ArrayBool_TO_ArrayByte(ADR(GVL_IO.Q_Temp),SIZEOF(GVL_IO.Q_Temp),ADR(GVL_IO.Q),SIZEOF(GVL_IO.Q));
ArrayByte_TO_ArrayBool(ADR(GVL_IO.I),SIZEOF(GVL_IO.I),ADR(GVL_IO.I_Temp),SIZEOF(GVL_IO.I_Temp));




// IO屏蔽
IF GVL_Data.stRecipe.eMachineType<>_eMachineType THEN
	_boolTemp:=ADR(GVL.stShield_I);
	FOR _i:=0 TO SIZEOF(GVL.stShield_I)-1 BY 1 DO
		_boolTemp[_i]:=FALSE;
	END_FOR
	_boolTemp:=ADR(GVL.stShield_Q);
	FOR _i:=0 TO SIZEOF(GVL.stShield_Q)-1 BY 1 DO
		_boolTemp[_i]:=FALSE;
	END_FOR
	_eMachineType:=GVL_Data.stRecipe.eMachineType;
END_IF



CASE GVL_Data.stRecipe.eMachineType OF
	E_MachineType._200:
		GVL.stShield_I[0,5]:=TRUE;		
		GVL.stShield_I[0,6]:=TRUE;		
		GVL.stShield_I[0,7]:=TRUE;		
		GVL.stShield_I[0,8]:=TRUE;		
		GVL.stShield_I[0,9]:=TRUE;		
		GVL.stShield_I[0,10]:=TRUE;		
		GVL.stShield_I[0,11]:=TRUE;		
		GVL.stShield_I[0,12]:=TRUE;	
		GVL.stShield_I[3,10]:=TRUE;
		GVL.stShield_I[3,11]:=TRUE;
		GVL.stShield_I[3,12]:=TRUE;
		GVL.stShield_I[3,13]:=TRUE;
		GVL.stShield_I[6,14]:=TRUE;
		
		GVL.stShield_Q[0,7]:=TRUE;
		GVL.stShield_Q[0,12]:=TRUE;
		GVL.stShield_Q[0,13]:=TRUE;
		GVL.stShield_Q[3,10]:=TRUE;
		GVL.stShield_Q[3,11]:=TRUE;
		GVL.stShield_Q[3,12]:=TRUE;
		GVL.stShield_Q[3,13]:=TRUE;
		GVL.stShield_Q[5,11]:=TRUE;
		
		FOR _i:=0 TO 15 BY 1 DO
			GVL.stShield_I[7,_i]:=TRUE;
			GVL.stShield_Q[6,_i]:=TRUE;
		END_FOR
	E_MachineType._367:
		FOR _i:=6 TO 15 BY 1 DO
			GVL.stShield_I[1,_i]:=TRUE;
			GVL.stShield_Q[1,_i]:=TRUE;
		END_FOR
	
		GVL.stShield_I[0,5]:=TRUE;		
		GVL.stShield_I[0,6]:=FALSE;		
		GVL.stShield_I[0,7]:=TRUE;				
		GVL.stShield_I[0,10]:=TRUE;		
		GVL.stShield_I[0,11]:=TRUE;		
		GVL.stShield_I[0,12]:=FALSE;	
		GVL.stShield_I[0,13]:=TRUE;
		GVL.stShield_I[0,14]:=TRUE;
		GVL.stShield_I[0,15]:=TRUE;
		GVL.stShield_I[3,14]:=TRUE;
		GVL.stShield_I[3,15]:=TRUE;
		GVL.stShield_I[4,0]:=TRUE;
		GVL.stShield_I[4,1]:=TRUE;
		GVL.stShield_I[6,3]:=TRUE;
		GVL.stShield_I[6,4]:=TRUE;
		GVL.stShield_I[5,6]:=TRUE;
		GVL.stShield_I[5,7]:=TRUE;
		GVL.stShield_I[5,8]:=TRUE;
		GVL.stShield_I[5,9]:=TRUE;
		GVL.stShield_I[5,10]:=TRUE;
		GVL.stShield_I[5,11]:=TRUE;
		GVL.stShield_I[5,12]:=TRUE;
		GVL.stShield_I[5,13]:=TRUE;
		GVL.stShield_I[5,14]:=TRUE;
		GVL.stShield_I[5,15]:=TRUE;
		GVL.stShield_I[6,13]:=TRUE;
		GVL.stShield_I[6,14]:=TRUE;
		
		GVL.stShield_Q[0,7]:=TRUE;
		GVL.stShield_Q[0,14]:=TRUE;
		GVL.stShield_Q[0,15]:=TRUE;
		GVL.stShield_Q[3,14]:=TRUE;
		GVL.stShield_Q[3,15]:=TRUE;
		GVL.stShield_Q[4,0]:=TRUE;
		GVL.stShield_Q[4,1]:=TRUE;
		GVL.stShield_Q[5,6]:=TRUE;
		GVL.stShield_Q[5,7]:=TRUE;
		GVL.stShield_Q[5,11]:=TRUE;
		GVL.stShield_Q[5,12]:=TRUE;
		GVL.stShield_Q[5,13]:=TRUE;
		GVL.stShield_Q[5,14]:=TRUE;
		GVL.stShield_Q[5,15]:=TRUE;
		
		FOR _i:=0 TO 15 BY 1 DO
			GVL.stShield_I[7,_i]:=TRUE;
			GVL.stShield_Q[6,_i]:=TRUE;
		END_FOR
	E_MachineType._373:
		GVL.stShield_I[0,5]:=TRUE;		
		GVL.stShield_I[0,6]:=TRUE;		
		GVL.stShield_I[0,7]:=TRUE;		
		GVL.stShield_I[0,8]:=TRUE;		
		GVL.stShield_I[0,9]:=TRUE;		
		GVL.stShield_I[0,10]:=TRUE;		
		GVL.stShield_I[0,11]:=TRUE;		
		GVL.stShield_I[0,12]:=TRUE;	
		GVL.stShield_I[0,13]:=FALSE;	
		GVL.stShield_I[0,14]:=FALSE;	
		GVL.stShield_I[0,15]:=FALSE;	
		GVL.stShield_I[2,0]:=TRUE;
		GVL.stShield_I[2,1]:=TRUE;
		GVL.stShield_I[2,4]:=TRUE;
		GVL.stShield_I[2,5]:=TRUE;
		GVL.stShield_I[3,0]:=TRUE;
		GVL.stShield_I[3,1]:=TRUE;
		GVL.stShield_I[3,10]:=TRUE;
		GVL.stShield_I[3,11]:=TRUE;
		GVL.stShield_I[3,12]:=TRUE;
		GVL.stShield_I[3,13]:=TRUE;
		GVL.stShield_I[3,14]:=TRUE;
		GVL.stShield_I[3,15]:=TRUE;
		GVL.stShield_I[4,0]:=TRUE;
		GVL.stShield_I[4,1]:=TRUE;
		GVL.stShield_I[4,8]:=TRUE;
		GVL.stShield_I[4,9]:=TRUE;
		GVL.stShield_I[5,10]:=TRUE;
		GVL.stShield_I[5,11]:=TRUE;
		GVL.stShield_I[5,12]:=TRUE;
		GVL.stShield_I[5,13]:=TRUE;
		GVL.stShield_I[5,14]:=TRUE;
		GVL.stShield_I[5,15]:=TRUE;
		GVL.stShield_I[6,13]:=TRUE;
		GVL.stShield_I[6,14]:=FALSE;
		
		GVL.stShield_Q[0,7]:=TRUE;
		GVL.stShield_Q[0,12]:=TRUE;		
		GVL.stShield_Q[0,13]:=TRUE;
		GVL.stShield_Q[2,0]:=TRUE;
		GVL.stShield_Q[2,1]:=TRUE;
		GVL.stShield_Q[2,4]:=TRUE;
		GVL.stShield_Q[2,5]:=TRUE;				
		GVL.stShield_Q[3,0]:=TRUE;
		GVL.stShield_Q[3,1]:=TRUE;
		GVL.stShield_Q[3,10]:=TRUE;
		GVL.stShield_Q[3,11]:=TRUE;
		GVL.stShield_Q[3,12]:=TRUE;
		GVL.stShield_Q[3,13]:=TRUE;
		GVL.stShield_Q[3,14]:=TRUE;
		GVL.stShield_Q[3,15]:=TRUE;
		GVL.stShield_Q[4,0]:=TRUE;
		GVL.stShield_Q[4,1]:=TRUE;
		GVL.stShield_Q[4,8]:=TRUE;
		GVL.stShield_Q[4,9]:=TRUE;
		GVL.stShield_Q[5,11]:=TRUE;
		GVL.stShield_Q[5,12]:=TRUE;
		GVL.stShield_Q[5,13]:=TRUE;
		GVL.stShield_Q[5,14]:=TRUE;
		GVL.stShield_Q[5,15]:=TRUE;
		
		FOR _i:=0 TO 15 BY 1 DO
			GVL.stShield_I[7,_i]:=TRUE;
			GVL.stShield_Q[6,_i]:=TRUE;
		END_FOR
	E_MachineType._069:
		GVL.stShield_I[0,5]:=TRUE;		
		GVL.stShield_I[0,6]:=TRUE;		
		GVL.stShield_I[0,7]:=TRUE;		
		GVL.stShield_I[0,8]:=TRUE;		
		GVL.stShield_I[0,9]:=TRUE;		
		GVL.stShield_I[0,10]:=TRUE;		
		GVL.stShield_I[0,11]:=TRUE;		
		GVL.stShield_I[0,12]:=TRUE;	
		GVL.stShield_I[2,0]:=TRUE;
		GVL.stShield_I[2,1]:=TRUE;
		GVL.stShield_I[2,4]:=TRUE;
		GVL.stShield_I[2,5]:=TRUE;
		GVL.stShield_I[3,10]:=TRUE;
		GVL.stShield_I[3,11]:=TRUE;
		GVL.stShield_I[3,12]:=TRUE;
		GVL.stShield_I[3,13]:=TRUE;
		GVL.stShield_I[3,14]:=TRUE;
		GVL.stShield_I[3,15]:=TRUE;
		GVL.stShield_I[4,0]:=TRUE;
		GVL.stShield_I[4,1]:=TRUE;
		GVL.stShield_I[5,6]:=TRUE;
		GVL.stShield_I[5,7]:=TRUE;
		GVL.stShield_I[5,8]:=TRUE;
		GVL.stShield_I[5,9]:=TRUE;
		GVL.stShield_I[5,10]:=TRUE;
		GVL.stShield_I[5,11]:=TRUE;
		GVL.stShield_I[5,12]:=TRUE;
		GVL.stShield_I[5,13]:=TRUE;
		GVL.stShield_I[5,14]:=TRUE;
		GVL.stShield_I[5,15]:=TRUE;
		GVL.stShield_I[6,13]:=TRUE;
		GVL.stShield_I[6,14]:=TRUE;
		
		GVL.stShield_Q[0,7]:=TRUE;
		GVL.stShield_Q[0,12]:=TRUE;
		GVL.stShield_Q[0,13]:=TRUE;
		GVL.stShield_Q[2,0]:=TRUE;
		GVL.stShield_Q[2,1]:=TRUE;
		GVL.stShield_Q[2,4]:=TRUE;
		GVL.stShield_Q[2,5]:=TRUE;
		GVL.stShield_Q[3,10]:=TRUE;
		GVL.stShield_Q[3,11]:=TRUE;
		GVL.stShield_Q[3,12]:=TRUE;
		GVL.stShield_Q[3,13]:=TRUE;
		GVL.stShield_Q[3,14]:=TRUE;
		GVL.stShield_Q[3,15]:=TRUE;
		GVL.stShield_Q[4,0]:=TRUE;
		GVL.stShield_Q[4,1]:=TRUE;
		GVL.stShield_Q[5,11]:=TRUE;
		GVL.stShield_Q[5,12]:=TRUE;
		GVL.stShield_Q[5,13]:=TRUE;
		GVL.stShield_Q[5,14]:=TRUE;
		GVL.stShield_Q[5,15]:=TRUE;
	
		FOR _i:=0 TO 15 BY 1 DO
			GVL.stShield_I[7,_i]:=TRUE;
			GVL.stShield_Q[6,_i]:=TRUE;
		END_FOR
	E_MachineType._311:
		GVL.stShield_I[0,5]:=FALSE;		
		GVL.stShield_I[0,6]:=TRUE;		
		GVL.stShield_I[0,7]:=TRUE;		
		GVL.stShield_I[0,8]:=TRUE;		
		GVL.stShield_I[0,9]:=TRUE;		
		GVL.stShield_I[0,10]:=TRUE;		
		GVL.stShield_I[0,11]:=TRUE;		
		GVL.stShield_I[0,12]:=TRUE;
		GVL.stShield_I[2,0]:=TRUE;
		GVL.stShield_I[2,1]:=TRUE;
		GVL.stShield_I[2,4]:=TRUE;
		GVL.stShield_I[2,5]:=TRUE;	
		GVL.stShield_I[3,0]:=TRUE;
		GVL.stShield_I[3,1]:=TRUE;
		GVL.stShield_I[3,10]:=TRUE;
		GVL.stShield_I[3,11]:=TRUE;
		GVL.stShield_I[3,12]:=TRUE;
		GVL.stShield_I[3,13]:=TRUE;
		GVL.stShield_I[3,14]:=TRUE;
		GVL.stShield_I[3,15]:=TRUE;
		GVL.stShield_I[4,0]:=TRUE;
		GVL.stShield_I[4,1]:=TRUE;
		GVL.stShield_I[5,6]:=TRUE;
		GVL.stShield_I[5,7]:=TRUE;
		GVL.stShield_I[5,8]:=TRUE;
		GVL.stShield_I[5,9]:=TRUE;
		GVL.stShield_I[5,10]:=TRUE;
		GVL.stShield_I[5,11]:=TRUE;
		GVL.stShield_I[5,12]:=TRUE;
		GVL.stShield_I[5,13]:=TRUE;
		GVL.stShield_I[5,14]:=TRUE;
		GVL.stShield_I[5,15]:=TRUE;
		GVL.stShield_I[6,13]:=TRUE;
		GVL.stShield_I[6,14]:=TRUE;
		
		GVL.stShield_Q[0,7]:=TRUE;
		GVL.stShield_Q[0,12]:=TRUE;
		GVL.stShield_Q[0,13]:=TRUE;
		GVL.stShield_Q[2,0]:=TRUE;
		GVL.stShield_Q[2,1]:=TRUE;
		GVL.stShield_Q[2,4]:=TRUE;
		GVL.stShield_Q[2,5]:=TRUE;
		GVL.stShield_Q[3,0]:=TRUE;
		GVL.stShield_Q[3,1]:=TRUE;
		GVL.stShield_Q[3,10]:=TRUE;
		GVL.stShield_Q[3,11]:=TRUE;
		GVL.stShield_Q[3,12]:=TRUE;
		GVL.stShield_Q[3,13]:=TRUE;
		GVL.stShield_Q[3,14]:=TRUE;
		GVL.stShield_Q[3,15]:=TRUE;
		GVL.stShield_Q[4,0]:=TRUE;
		GVL.stShield_Q[4,1]:=TRUE;
		GVL.stShield_Q[5,11]:=TRUE;
		GVL.stShield_Q[5,12]:=TRUE;
		GVL.stShield_Q[5,13]:=TRUE;
		GVL.stShield_Q[5,14]:=TRUE;
		GVL.stShield_Q[5,15]:=TRUE;
END_CASE
END_ACTION

ACTION A_Line:
GVL.arrFbLine[E_LineAxis.Acquire](System:=G_stSystem , Moving=>GVL.Q.bAcquireAxis );
GVL.arrFbLine[E_LineAxis.UnloadForck](System:=G_stSystem , Moving=>GVL.Q.bUnloadFrock );
GVL.arrFbLine[E_LineAxis.UnloadUc](System:=G_stSystem , Moving=>GVL.Q.bUnloadUcAxis );
GVL.arrFbLine[E_LineAxis.Dismantling](System:=G_stSystem , Moving=>GVL.Q.bDismantlingAxis );
GVL.arrFbLine[E_LineAxis.AcquireFront](System:=G_stSystem , Moving=>GVL.Q.bAcquireFrontAxis );

IF G_stSystem.stMode.bAutoRunning THEN
	GVL.arrFbLine[E_LineAxis.Acquire].M_Jog(1);
	GVL.arrFbLine[E_LineAxis.UnloadForck].M_Jog(1);
	GVL.arrFbLine[E_LineAxis.Dismantling].M_Jog(1);
	GVL.arrFbLine[E_LineAxis.AcquireFront].M_Jog(1);
END_IF
END_ACTION

END_PROGRAM

(* stored: Version 1.1.0.1, ProductVersion 3.1.4024.3
   POU P_Device: Id {13cc3208-eb13-4248-ad09-86d2342ef435}, SpecialFunc None
   Action A_Axis: Id {ff47a3e6-d233-4182-ae50-c85a3b8a742d}
   Action A_Cylinder: Id {f287f90e-ded2-434e-9553-ff04ee696bc4}
   Action A_CylinderTest: Id {d6a0c848-c9af-4665-8eae-053e4364a902}
   Action A_CylinderTest069: Id {5bdd318a-afde-4f44-9b1c-1cf60fbe0dc0}
   Action A_CylinderTest201: Id {9f5fffe6-759d-43ec-9a2f-9aaa9b32cddf}
   Action A_CylinderTest311: Id {05f3ebc1-9597-4352-ab77-b74849cc9f67}
   Action A_CylinderTest367: Id {c9fd115b-a8aa-475c-a7d3-fd9552ad2280}
   Action A_CylinderTest373: Id {a87c1324-8fa2-4e8f-b6f4-e294dfa9223b}
   Action A_Info: Id {a7862511-5848-48f5-b27a-2def49c23547}
   Action A_InOut: Id {cd9529a3-874d-4a86-899b-b7fed3efd57b}
   Action A_Line: Id {17405297-3473-449e-8cdf-f5ce13cffb81} *)
